(* CODESYS project Uppgift 5.project

Project tree, tasks and I/O mapping:
  Device : CODESYS Control Win V3, 3S - Smart Software Solutions GmbH, order no. 305021, version 3.5.10.40
    application Application
      libraries: Standard, * (System)
      task MainTask (cyclic, interval t#20ms, priority 1) calls PLC_PRG
      task VISU_TASK (cyclic, interval 100 ms, priority 31) calls VisuElems.Visu_Prg
      program PLC_PRG [LD]
      global variables GVL
      visualisation VisualizationBTNLamp
  libraries: VisuSymbols, 3.5.10.0 (System)
  text list GlobalTextList
*)

// Device/Application/GVL
{attribute 'qualified_only'}
VAR_GLOBAL
	
END_VAR

// Device/Application/PLC_PRG
PROGRAM PLC_PRG
VAR
	Red_Btn: BOOL;
	Blue_Btn: BOOL;
	Green_lamp: BOOL;
	Blue_lamp: BOOL;
	Red_lamp: BOOL;
END_VAR

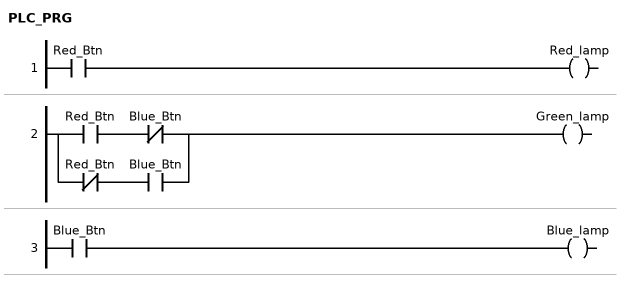
// NETWORK 1
Red_lamp := Red_Btn;

// NETWORK 2
Green_lamp := Red_Btn AND NOT Blue_Btn OR NOT Red_Btn AND Blue_Btn;

// NETWORK 3
Blue_lamp := Blue_Btn;

END_PROGRAM

// Device/Application/VisualizationBTNLamp
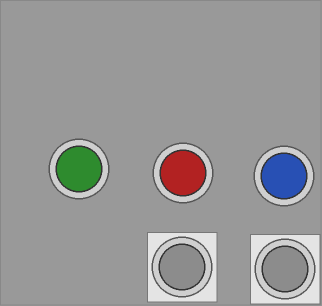
VISUALIZATION VisualizationBTNLamp  // 322x306
    Lamp1 (44,134 70x70), variable: PLC_PRG.Green_lamp, style: Lamp-Lamp1-Green
    Lamp1 (148,138 70x70), variable: PLC_PRG.Red_lamp, style: Lamp-Lamp1-Red
    Lamp1 (249,141 70x70), variable: PLC_PRG.Blue_lamp, style: Lamp-Lamp1-Blue
    PushSwitch (147,232 70x70), variable: PLC_PRG.Red_Btn, behaviour: TOGGLE, style: Switch-PushSwitch-Gray
    PushSwitch (250,234 70x70), variable: PLC_PRG.Blue_Btn, behaviour: TOGGLE, style: Switch-PushSwitch-Gray
END_VISUALIZATION
